Fanuc KAREL source: KT00366.KL

PROGRAM KT00366
%NOLOCKGROUP
VAR
  I1: INTEGER
  R2: REAL
  OUT: BOOLEAN
BEGIN
  I1 = 2
    R2 = 3.0
  OUT = I1 <= R2
END KT00366
